{attribute 'qualified_only'}
{attribute 'strict'}
TYPE eSCARATask :
(
	task_init := 0,
	task_regular_check_scara1 := 1,
	task_regular_check_scara2 := 2,
	task_assemble_scara1 := 3,
	task_snap_scara2 := 4,
	task_load_drop :=5
) INT;
END_TYPE

(* stored: Version 1.1.0.1, ProductVersion 3.1.4024.0
   EnumerationTextList eSCARATask: Id {f8c2628f-ecab-4dc2-b5c4-01c824186724} *)
